{attribute 'no_explicit_call' := 'do not call this POU directly'} 
FUNCTION_BLOCK PUBLIC FB_ListTestsuite IMPLEMENTS I_ListTestsuite
VAR
	pList: 			POINTER TO I_Testsuite;
	nLength:		DINT;
	aList:			POINTER TO POINTER TO ARRAY [0..100] OF I_Testsuite:=ADR(pList);
END_VAR

METHOD FB_exit : BOOL
VAR_INPUT
	bInCopyCode : BOOL; // if TRUE, the exit method is called for exiting an instance that is copied afterwards (online change).
END_VAR
M_Clear();
END_METHOD

METHOD M_Add : BOOL
VAR_INPUT
	Testsuite: 	I_Testsuite;
END_VAR
VAR
	pOldList: 	POINTER TO I_Testsuite;
END_VAR
IF Testsuite <> 0 THEN
	// First Item
	IF pList = 0 THEN
		nLength:= nLength + 1;
		pList:= __NEW(POINTER TO I_Testsuite,DINT_TO_UDINT(nLength));
	ELSE
		// Item already in List
		IF M_Search(Testsuite) = -1 THEN
			// backup 
			pOldList:= pList;
			// new Length
			nLength:= nLength + 1;
			// new pointer
			pList:= __NEW(POINTER TO I_Testsuite,DINT_TO_UDINT(nLength));
			// restore
			Memcpy(pList,pOldList, SIZEOF(POINTER TO I_Testsuite)*DINT_TO_UDINT(nLength -1));
			// delete old
			__DELETE(pOldList);
		ELSE
			M_Add:= FALSE;	
			RETURN;
		END_IF
	END_IF
	// add new Object
	pList[nLength-1]:= Testsuite;
	M_Add:= TRUE;
ELSE
	M_Add:= FALSE;	
END_IF
END_METHOD

METHOD M_Clear
IF pList <> 0 THEN
	nLength:= 0;
	__DELETE(pList);
END_IF
END_METHOD

METHOD M_Get : I_Testsuite
VAR_INPUT
	Index: 	DINT;
END_VAR
IF Index <= nLength THEN
	M_Get:= pList[Index];
END_IF
END_METHOD

METHOD M_Index : DINT
VAR_INPUT
	Testsuite: 	I_Testsuite;
END_VAR
VAR
	nIndex: 	DINT;
END_VAR
// Object already in List
M_Index := -1;
WHILE nIndex < nLength DO
    IF (pList[nIndex] = Testsuite) THEN
        M_Index := nIndex;
        RETURN;
    END_IF
	nIndex := nIndex + 1;
END_WHILE
END_METHOD

METHOD M_Remove : BOOL
VAR_INPUT
	Testsuite: 			I_Testsuite;
END_VAR
VAR
	pOldList:			POINTER TO I_Testsuite;
	nPosition: 			DINT;
END_VAR
IF Testsuite <> 0 THEN
	// First Item
	IF nLength >= 0 THEN
		// Item already in List
		nPosition:= M_Search(Testsuite);
		IF nPosition <> -1 THEN
			// backup 
			pOldList:= pList;
			// new Length
			nLength:= nLength -1;
			// new pointer
			pList:= __NEW(POINTER TO I_Testsuite,DINT_TO_UDINT(nLength));
			// restore lower part
			Memcpy(pList,pOldList, SIZEOF(POINTER TO I_Testsuite) * DINT_TO_UDINT(nPosition));
			//pList[nPosition]:= iObject;
			Memcpy(pList + (SIZEOF(POINTER TO I_Testsuite)*nPosition),pOldList + (SIZEOF(POINTER TO I_Testsuite)*(nPosition + 1)), SIZEOF(POINTER TO I_Testsuite) * DINT_TO_UDINT(nLength - nPosition));
			// delete old
			__DELETE(pOldList);
		ELSE
			M_Remove:= FALSE;	
			RETURN;
		END_IF
	ELSE
		M_Remove:= FALSE;	
		RETURN;
	END_IF
	M_Remove:= TRUE;
ELSE
	M_Remove:= FALSE;	
END_IF
END_METHOD

METHOD M_Search : DINT
VAR_INPUT
	Testsuite: 	I_Testsuite;
END_VAR
VAR
	nIndex: 	UINT;
END_VAR
// Object already in List
M_Search := -1;
WHILE nIndex < nLength DO
    IF (pList[nIndex] = Testsuite) THEN
        M_Search := nIndex;
        RETURN;
    END_IF
	nIndex := nIndex + 1;
END_WHILE
END_METHOD

PROPERTY P_Length : DINT
GET
P_Length:= nLength;
END_GET
END_PROPERTY

END_FUNCTION_BLOCK

(* stored: Version 1.1.0.1
   POU FB_ListTestsuite: Id {80a15822-49de-454f-b0fc-12851675b870}, SpecialFunc None
   Method FB_exit: Id {206ba99c-f43a-4ef7-9ab3-3aa10406299c}
   Method M_Add: Id {a38c7fef-d96a-4183-97fc-f0e5fdcf0ccf}
   Method M_Clear: Id {bb7164ec-9ad3-43d2-bddd-bf3368367664}
   Method M_Get: Id {d9624459-7fd8-4784-aea6-5c773f6a64a0}
   Method M_Index: Id {a8754c07-7f0e-4184-834d-318ea0557896}
   Method M_Remove: Id {e3d569c0-1249-4bbc-9b3c-c9d8221349af}
   Method M_Search: Id {b4574359-c512-4073-955e-3a3fc1e43b2b}
   Property P_Length: Id {0b018640-abb2-489d-958f-1e0d7c39741f}
   Get Get: Id {394102f8-8cf0-4f3e-a868-8eb035088153} *)
